// TIA Portal V19 export
TYPE "Alarm_Parameter"
   STRUCT
      nicht_Hupe_Rot : Bool;   // Standardmässig immer Rot, einschalten wenn nicht gewünscht
      Hupe_Gelb : Bool;
      Hupe_Blau : Bool;
      Hupe_Dauer_Rot : Bool;
      Hupe_Dauer_Gelb : Bool;
      Hupe_Dauer_Blau : Bool;
      nicht_La_Rot : Bool;   // Standardmässig immer Rot, einschalten wenn nicht gewünscht
      La_Gelb : Bool;
      La_Blau : Bool;
      La_Quit_Err : Bool;
   END_STRUCT;
END_TYPE
